FUNCTION FUN_Substract : REAL
VAR_INPUT
		f_Inp1			: REAL;
		f_Inp2			: REAL;
END_VAR
VAR
END_VAR

FUN_Substract := f_Inp1 - f_Inp2;

END_FUNCTION

(* stored: Version 1.1.0.1, ProductVersion 3.1.4024.9
   POU FUN_Substract: Id {255bd7b1-456b-4cd3-8f01-558326a1c67c}, SpecialFunc None *)
